INTERFACE ITF_MechanischeRem

PROPERTY ActueleRemStand : BOOL
GET
END_GET
END_PROPERTY

METHOD RemLos
END_METHOD

METHOD RemVast
VAR_INPUT
END_VAR
END_METHOD

PROPERTY VerwachteRemStand : BOOL
GET
END_GET
SET
END_SET
END_PROPERTY

END_INTERFACE

(* stored: Version 1.1.0.1
   Itf ITF_MechanischeRem: Id {bc04c6e4-218a-41e4-a45e-c4d57f019239}
   Folder Methods: Id {17035f7d-6cfb-4ea6-a1b0-54d87b4cb342}
   Folder Properties: Id {76cdae90-1f72-4916-b040-1b60d4fd2242}
   Property ActueleRemStand: Id {5cf25cdf-dc7d-496c-9269-62220177bb71}
   Get Get: Id {f53046ea-8b62-414b-a7a5-d7aa3fac9cdd}
   Method RemLos: Id {8fc0ebcb-ba83-46a2-b549-645ec2d8bb5d}
   Method RemVast: Id {62a87b0c-c27e-4937-8362-11ed627c827b}
   Property VerwachteRemStand: Id {61cd89cd-32c1-401f-8f8e-d9d3ae767082}
   Get Get: Id {256e4e51-fdc5-47db-b94c-1c3fe58d28e0}
   Set Set: Id {4ccc1dc8-1d60-4360-b281-31f559dcafd6} *)
